FUNCTION_BLOCK EL4031
VAR
	_io : EL4xx1_Data;
	{attribute addProperty Name "WcState"}
	_wcState : WcStateBase;
	{attribute addProperty Name "Info data"}
	_infoData : InfoDataAds;
END_VAR

PROPERTY IO : REFERENCE TO EL4xx1_Data
GET
IO REF= _io;
END_GET
END_PROPERTY

PROPERTY WcState : REFERENCE TO WcStateBase
GET
WcState REF= _wcState;
END_GET
END_PROPERTY

END_FUNCTION_BLOCK

(* stored: Version 1.1.0.1, ProductVersion 3.1.4024.9
   POU EL4031: Id {667b1c07-9866-0169-2624-25728cd2baad}, SpecialFunc None
   Property IO: Id {3566ffd6-3143-0397-24fd-22aae1377d13}
   Get Get: Id {f9da71bc-7159-0276-2a37-ce6d12a4da4a}
   Property WcState: Id {6c34aad5-c454-0b2e-2042-1a2fbb562e7a}
   Get Get: Id {64074e6c-6a58-0c05-3300-c1aab67f2cb1} *)
